FUNCTION IsValidProperty : BOOL
VAR_INPUT
	PropertyToCheck : I_Parameter;
END_VAR

IsValidProperty := PropertyToCheck <> 0;

END_FUNCTION

(* stored: Version 1.1.0.1, ProductVersion 3.1.4024.12
   POU IsValidProperty: Id {f27cfd1a-d935-0531-0f17-a6712ace4c45}, SpecialFunc None *)
